PROGRAM Axis_1
VAR
    bLimitPowerAxis1 AT %Q*: BOOL := TRUE;
END_VAR
VAR // added by the converter: edge detectors and wires of the graphical bodies
    _w1, _w2 : BOOL;
END_VAR

//Initial parameters of an Axis
IF _TaskInfo[fbGetCurTaskIndex.index].FirstCycle THEN
    //Initial default values:
    GVL.astAxes[1].stConfig.eHomeSeq := 0;
    GVL.astAxes[1].stConfig.fHomePosition := 0.0;
    GVL.astAxes[1].stConfig.fHomeFinishDistance := 0.0;
END_IF

ACT_1_Interlock();

// Brake control from GUI
main.stHWStatusX.bBrakeReleased:=main.stHWControlX.bBrakeReleaseCmd;

// Enable Cmd from GUI
GVL.astAxes[1].stControl.bEnable:=main.stHWControlX.bEnable;
main.stHWStatusX.bEnabled:=GVL.astAxes[1].stStatus.bEnabled;

// Trigger Abs movement from GUI
IF main.stHWControlX.bExecuteAbsPos  AND NOT GVL.astAxes[1].stStatus.bBusy THEN
  GVL.astAxes[1].stControl.eCommand:=E_MotionFunctions.eMoveAbsolute;
  GVL.astAxes[1].stControl.bExecute:=TRUE;
  main.stHWControlX.bExecuteAbsPos:=FALSE;
END_IF

// Trigger Const Velo movement from GUI
IF main.stHWControlX.bExecuteConstVelo AND NOT GVL.astAxes[1].stStatus.bBusy THEN
  GVL.astAxes[1].stControl.eCommand:=E_MotionFunctions.eMoveVelocity;
  GVL.astAxes[1].stControl.bExecute:=TRUE;
  main.stHWControlX.bExecuteConstVelo:=FALSE;
END_IF

// Trigger Home vs LimitFwd (should be valid for all axes) from GUI
IF main.stHWControlX.bExecuteHome  AND NOT GVL.astAxes[1].stStatus.bBusy THEN
  GVL.astAxes[1].stConfig.fHomingVelFromCam:=GVL_Parameters.fXHomeVelOffCam;
  GVL.astAxes[1].stConfig.fHomingVelToCam:=GVL_Parameters.fXHomeVelToCam;
  GVL.astAxes[1].stConfig.fHomePosition:=GVL_Parameters.fXHomePosition;
  GVL.astAxes[1].stControl.eCommand:=E_MotionFunctions.eHome;
  GVL.astAxes[1].stConfig.eHomeSeq:=E_HomingRoutines.eHomeToLimit_Fwd;
  GVL.astAxes[1].stControl.bExecute:=TRUE;
  main.stHWControlX.bExecuteHome:=FALSE;
END_IF

//Stop Motion from GUI
IF main.stHWControlX.bExecuteStop THEN
  GVL.astAxes[1].stControl.bStop := NOT(GVL.astAxes[1].stControl.bStop);
  GVL.astAxes[1].stControl.bExecute:=FALSE;
  main.stHWControlX.bExecuteStop:=FALSE;
END_IF

// Error Code
GVL.astAxes[1].stStatus.nErrorID;

main.stHWStatusX.bBusy:=GVL.astAxes[1].stStatus.bBusy;
GVL.astAxes[1].stControl.bReset:=main.stHWControlX.bExecuteReset;
main.stHWControlX.bExecuteReset:=FALSE;
main.stHWStatusX.bHomed:=GVL.astAxes[1].stStatus.bHomed;
main.stHWStatusX.bHomingCmdActive:=GVL.astAxes[1].stControl.eCommand=E_MotionFunctions.eHome AND 
                                   GVL.astAxes[1].stConfig.eHomeSeq=E_HomingRoutines.eHomeToLimit_Fwd;

// Hard code velocities and acc/dec
GVL.astAxes[1].stControl.fAcceleration:=GVL_Parameters.fXStepperTargetAcc;
GVL.astAxes[1].stControl.fDeceleration:=GVL_Parameters.fXStepperTargetAcc;
GVL.astAxes[1].stControl.fVelocity:=GVL_Parameters.fXStepperTargetVelo;

// Check position is inside limits (and homed)
main.stHWStatusX.bLoLoAlm:=gvl.astAxes[1].stStatus.fActPosition < GVL_Parameters.fXRangeL2 OR NOT main.stHWStatusX.bHomed;
main.stHWStatusX.bLoAlm:=gvl.astAxes[1].stStatus.fActPosition < GVL_Parameters.fXRangeL1 OR NOT main.stHWStatusX.bHomed;
main.stHWStatusX.bHiAlm:=gvl.astAxes[1].stStatus.fActPosition > GVL_Parameters.fXRangeH1 OR NOT main.stHWStatusX.bHomed;
main.stHWStatusX.bhiHiAlm:=gvl.astAxes[1].stStatus.fActPosition > GVL_Parameters.fXRangeH2 OR NOT main.stHWStatusX.bHomed;

ACTION ACT_1_Interlock:
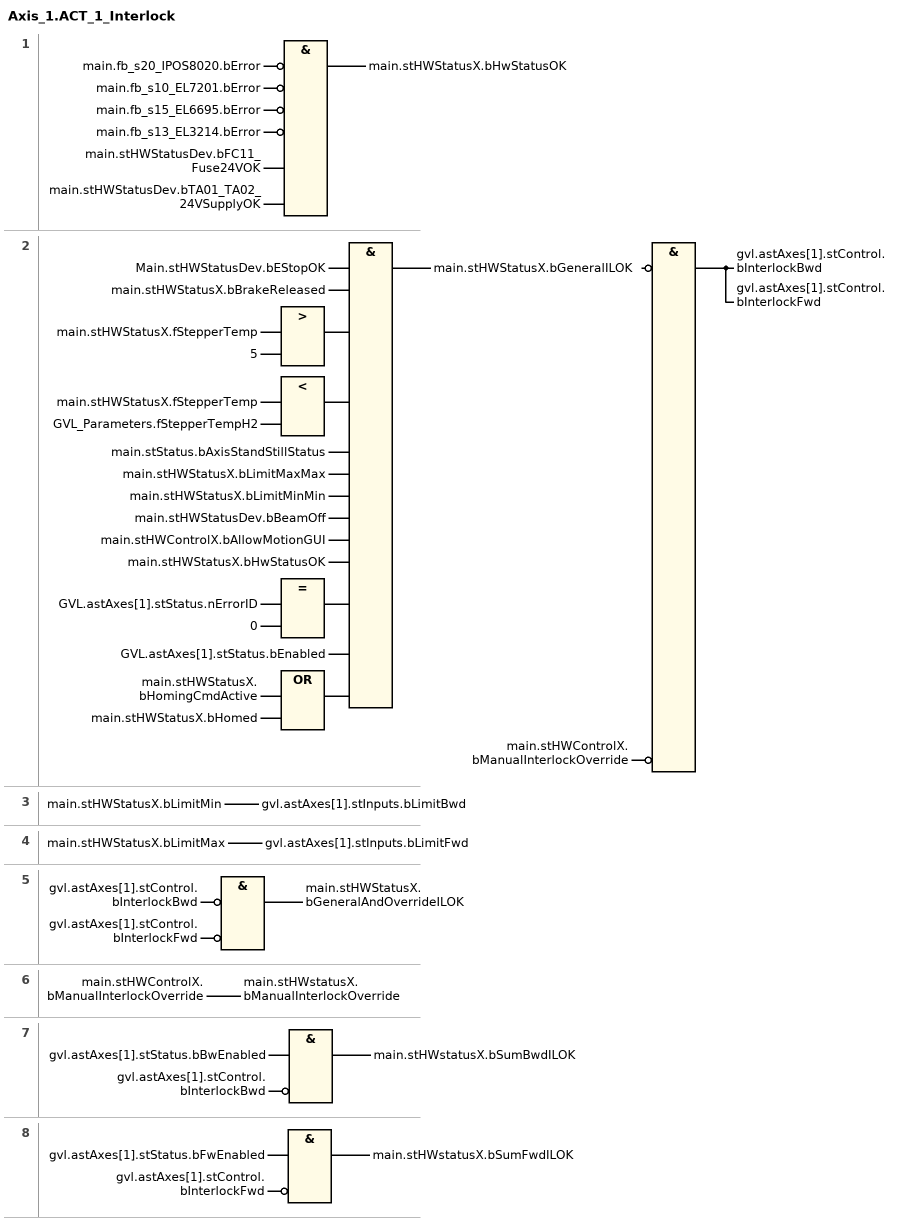
// NETWORK 1
main.stHWStatusX.bHwStatusOK := NOT main.fb_s20_IPOS8020.bError AND NOT main.fb_s10_EL7201.bError AND NOT main.fb_s15_EL6695.bError AND NOT main.fb_s13_EL3214.bError AND main.stHWStatusDev.bFC11_Fuse24VOK AND main.stHWStatusDev.bTA01_TA02_24VSupplyOK;

// NETWORK 2
_w1 := Main.stHWStatusDev.bEStopOK AND main.stHWStatusX.bBrakeReleased AND main.stHWStatusX.fStepperTemp > 5 AND main.stHWStatusX.fStepperTemp < GVL_Parameters.fStepperTempH2 AND main.stStatus.bAxisStandStillStatus AND main.stHWStatusX.bLimitMaxMax AND main.stHWStatusX.bLimitMinMin AND main.stHWStatusDev.bBeamOff AND main.stHWControlX.bAllowMotionGUI AND main.stHWStatusX.bHwStatusOK AND GVL.astAxes[1].stStatus.nErrorID = 0 AND GVL.astAxes[1].stStatus.bEnabled AND (main.stHWStatusX.bHomingCmdActive OR main.stHWStatusX.bHomed);
main.stHWStatusX.bGeneralILOK := _w1;
_w2 := NOT _w1 AND NOT main.stHWControlX.bManualInterlockOverride;
gvl.astAxes[1].stControl.bInterlockBwd := _w2;
gvl.astAxes[1].stControl.bInterlockFwd := _w2;

// NETWORK 3
gvl.astAxes[1].stInputs.bLimitBwd := main.stHWStatusX.bLimitMin;

// NETWORK 4
gvl.astAxes[1].stInputs.bLimitFwd := main.stHWStatusX.bLimitMax;

// NETWORK 5
main.stHWStatusX.bGeneralAndOverrideILOK := NOT gvl.astAxes[1].stControl.bInterlockBwd AND NOT gvl.astAxes[1].stControl.bInterlockFwd;

// NETWORK 6
main.stHWstatusX.bManualInterlockOverride := main.stHWControlX.bManualInterlockOverride;

// NETWORK 7
main.stHWstatusX.bSumBwdILOK := gvl.astAxes[1].stStatus.bBwEnabled AND NOT gvl.astAxes[1].stControl.bInterlockBwd;

// NETWORK 8
main.stHWstatusX.bSumFwdILOK := gvl.astAxes[1].stStatus.bFwEnabled AND NOT gvl.astAxes[1].stControl.bInterlockFwd;
END_ACTION

END_PROGRAM

(* stored: Version 1.1.0.1, ProductVersion 3.1.4024.6
   POU Axis_1: Id {734d3f4c-c951-47c9-b623-1f718ea980b1}, SpecialFunc None
   Action ACT_1_Interlock: Id {ca43ea7f-b212-458e-a066-b237d81a70c7} *)
